Staubli VAL3: iLevel3.pgx

public program iLevel3(num& nNum[] (dimensions=1))
begin
  nNum=dioGet(iLevel3)
end
